PROGRAM MAIN
VAR
END_VAR

END_PROGRAM

(* stored: Version 1.1.0.1, ProductVersion 3.1.4026.6
   POU MAIN: Id {02b73f09-8514-42a5-a804-e614cbd39f48}, SpecialFunc None *)
